FUNCTION_BLOCK FB_Object
VAR_INPUT
END_VAR
VAR_OUTPUT
END_VAR
VAR
	nObjectID			: UINT;
	eObjectType 		: E_ObjectType;
	eObjectGroup		: E_ObjectGroup;//Zugehörigkeit zu Objektgruppe [Flags]
	pObjCollectNode		: POINTER TO FB_ObjCollectionNode;
	pParentSlot			: POINTER TO FB_Slot;
	nNoOfProps			: UINT;
	wChecksum			: WORD;
END_VAR

//Basisklasse für alle Objekte

METHOD M_AddChild : ERRORID
VAR_INPUT
	pObject	: POINTER TO FB_Object;
	nSlotNr	: UINT;
	nIndex : INT;
END_VAR
END_METHOD

METHOD M_bIsGroup : BOOL
VAR_INPUT
	eGroup	: E_ObjectGroup;
END_VAR
M_bIsGroup := (eObjectGroup AND eGroup) = eGroup;
END_METHOD

METHOD M_CheckProps : ERRORID
END_METHOD

METHOD M_ClearAllProps

VAR_INPUT
	bIgnoreParent : BOOL; //Es wird das gesamte OD gelöscht. -> Zeiger auf Parent nicht mehr gültig!
END_VAR
END_METHOD

METHOD M_GetAllProps : ERRORID
VAR_INPUT
	refCmdData	: REFERENCE TO ST_CmdData;
END_VAR
END_METHOD

METHOD M_GetDevice : I_Device
VAR_INPUT
END_VAR
END_METHOD

METHOD M_GetPropCheckSum : UINT
VAR_INPUT
END_VAR

VAR
	i			: UINT;
	stData 		: ST_CmdData;
END_VAR
M_GetAllProps(stData);
wChecksum := F_DATA_TO_CRC16_CCITT(ADR(stData.n32Data[0]),nNoOfProps * 4,16#FFFF);
M_GetPropCheckSum := wChecksum;
END_METHOD

METHOD M_GetSlot : POINTER TO FB_Slot
VAR_INPUT
	nSlotNr : UINT;
END_VAR
END_METHOD

METHOD M_GetSlotFromChild : POINTER TO FB_Slot
VAR_INPUT
	pObject : POINTER TO FB_Object;
END_VAR
END_METHOD

METHOD M_RemoveChild : ERRORID
VAR_INPUT
	pObject	: POINTER TO FB_Object;
END_VAR

VAR
	iter : FB_ObjCollectIterator;
END_VAR
//Das Objekt in der Collection suchen (flach)
pObjCollectNode^.nodes.M_GetIterator(iter);
WHILE iter.pNode > 0 DO
	IF iter.pNode^.P_pObject = pObject THEN
		//Falls Object an einem Slot, von diesem entfernen
		IF pObject^.P_pParentSlot > 0 THEN
			pObject^.P_pParentSlot^.P_pChild := 0;
		END_IF
		pObjCollectNode^.nodes.M_RemoveNode(iter.pNode);
		pObject^.M_UpdateParent();
		EXIT;
	END_IF
	iter.M_Increment();
END_WHILE

IF iter.pNode = 0 THEN
	M_RemoveChild := E_ErrorIdObjMgmt.ERRORID_ObjectNotInCollection;
END_IF
END_METHOD

METHOD M_SetAllProps : ERRORID
VAR_INPUT
	refCmdData	: REFERENCE TO ST_CmdData;
END_VAR
END_METHOD

METHOD M_SetSingleProp : ERRORID
VAR_INPUT
	refCmdData	: REFERENCE TO ST_CmdData;
END_VAR
END_METHOD

METHOD M_UpdateParent
END_METHOD

PROPERTY P_bHasChilds : BOOL
GET
P_bHasChilds := pObjCollectNode > 0 and_then pObjCollectNode^.nodes.nCount > 0;
END_GET
END_PROPERTY

PROPERTY P_eObjectGroup : E_ObjectGroup
GET
P_eObjectGroup := eObjectGroup;
END_GET
END_PROPERTY

PROPERTY P_eObjectType : E_ObjectType
GET
P_eObjectType := eObjectType;
END_GET
END_PROPERTY

PROPERTY P_nNoOfProps : UINT
GET
P_nNoOfProps := nNoOfProps;
END_GET
END_PROPERTY

PROPERTY P_nNotifyId : UINT
GET
END_GET
SET
END_SET
END_PROPERTY

PROPERTY P_nObjectID : UINT
GET
P_nObjectID := nObjectID;
END_GET
SET
nObjectID := P_nObjectID;
END_SET
END_PROPERTY

PROPERTY P_nParentSlotNr : UINT
GET
IF pParentSlot > 0 THEN
	P_nParentSlotNr := pParentSlot^.P_nNr;
END_IF
END_GET
END_PROPERTY

PROPERTY P_pObjCollectNode : POINTER TO FB_ObjCollectionNode
GET
P_pObjCollectNode := pObjCollectNode;
END_GET
SET
pObjCollectNode := P_pObjCollectNode;
END_SET
END_PROPERTY

PROPERTY P_pParentObject : POINTER TO FB_Object
GET
IF pObjCollectNode > 0 AND_THEN pObjCollectNode^.pOwnerColl > 0 AND_THEN pObjCollectNode^.pOwnerColl^.pOwnerNode > 0 THEN
	P_pParentObject := pObjCollectNode^.pOwnerColl^.pOwnerNode^.P_pObject;
END_IF
END_GET
END_PROPERTY

PROPERTY P_pParentSlot : POINTER TO FB_Slot
GET
P_pParentSlot := pParentSlot;
END_GET
END_PROPERTY

END_FUNCTION_BLOCK

(* stored: Version 1.1.0.1
   POU FB_Object: Id {dafb0000-3307-4ea2-a148-e6eeb646c546}, SpecialFunc None
   Method M_AddChild: Id {15681bd5-aa3d-4151-93a8-ef366c5b3c5e}
   Method M_bIsGroup: Id {148466bb-7554-4bd2-af99-8b6e209359f3}
   Method M_CheckProps: Id {e299850d-443c-4f77-9a4b-a14f1f4e80ae}
   Method M_ClearAllProps: Id {c6181026-0c4e-40e4-bd77-8cec92305f9e}
   Method M_GetAllProps: Id {3ba8a592-fc8f-4794-9a6e-03bbd147e4ea}
   Method M_GetDevice: Id {0c76071d-8fd4-4334-993f-7de7f1da8394}
   Method M_GetPropCheckSum: Id {1b864eb4-ca15-4169-88ba-ca0b087c5b80}
   Method M_GetSlot: Id {ba9bed8b-d5e7-476f-9359-48c995c9302a}
   Method M_GetSlotFromChild: Id {8851af2f-0e6f-4d0a-81d3-b945a799be53}
   Method M_RemoveChild: Id {a4fdd1a9-85af-4d60-804f-2b95973c7db4}
   Method M_SetAllProps: Id {2aa1fadb-c8f5-4fab-a5d0-64328a4d0239}
   Method M_SetSingleProp: Id {bd51375e-f7d7-466b-9ea7-2f695e193e51}
   Method M_UpdateParent: Id {60a3d0a9-4998-4589-a7d6-89641a375343}
   Property P_bHasChilds: Id {ace6323d-7d9d-4d1f-8e5b-a91592ab1a10}
   Get Get: Id {8afe265b-2f92-4dbe-9ff3-6a6f4c11b095}
   Property P_eObjectGroup: Id {b94e65bd-d653-427d-8fa5-6193a0e4b5f5}
   Get Get: Id {ea5ad8b5-52a1-42df-ab1a-bc744dff3896}
   Property P_eObjectType: Id {61c4d3a3-c06f-49c9-83a6-d9c40a7b9275}
   Get Get: Id {669098f0-4ac6-42ab-996d-03def5965c2b}
   Property P_nNoOfProps: Id {7b3ff459-ce45-4ac3-b566-241558331cbf}
   Get Get: Id {f81fe8ac-9e2d-4b54-803f-ffcc2e7cb497}
   Property P_nNotifyId: Id {e4b2e2df-1801-4f89-8df1-7548bac25d8c}
   Get Get: Id {aa02bafe-4392-46db-ad39-296675877b46}
   Set Set: Id {c1c872a4-bc23-44cd-946e-07cc3255a58b}
   Property P_nObjectID: Id {edd2a331-c397-4992-b113-832f9415bd91}
   Get Get: Id {180a3d84-00f7-48f6-9df8-142b6f1bf69a}
   Set Set: Id {1c81fe87-3942-4c0d-b798-a6c36cb387d7}
   Property P_nParentSlotNr: Id {80aadf76-7e96-40d5-9b64-f68bbc8e10de}
   Get Get: Id {2e344dce-1eec-4b50-b4e0-7384751712c5}
   Property P_pObjCollectNode: Id {44c81f7b-fdd1-401c-99b9-979d769599c9}
   Get Get: Id {3845ab7e-2398-4bcb-bea9-d268027aa224}
   Set Set: Id {dc96722f-4bc7-469f-9085-bc5ba8afd212}
   Property P_pParentObject: Id {4c243c53-27fd-4f6e-a2e8-ed45a2496a0d}
   Get Get: Id {b2175f77-e943-4cdd-a82a-2897c541a222}
   Property P_pParentSlot: Id {f8ea0287-83ca-4904-9770-3f0dcbd44ea6}
   Get Get: Id {619f79e0-a1c7-48b9-b1d4-17012cfa4233} *)
